
TYPE "DriveControllerOutput"
STRUCT
        status : WORD;
        errorStatus : WORD;
        actualSpeed : INT;
        isRunning : BOOL;
        isSafetyActive : BOOL;
        runtime : INT;
        speedHistory : ARRAY[0..9] OF INT;
END_STRUCT;
END_TYPE